{attribute 'qualified_only'}
VAR_GLOBAL
END_VAR

(* stored: Version 1.1.0.1, ProductVersion 3.1.4024.12
   GVL G_Input: Id {60f3cd38-efe2-49f3-9587-01cf731da48b} *)
